FUNCTION_BLOCK COLORSENSOR_MDL (* Color sensor model *)
  (* Standard: 61499-2 *)
  (* Version 0.3, 2009-09-15, JHC, Holobloc Inc, Changed transition priorities. *)
  (* Version 0.2, 2003-12-04, JHC, Rockwell Automation, Renamed for better indexing. *)
  (* Version 0.1, 2002-11-05, JHC, Rockwell Automation, Corrected missing ST element in Algorithm REQ. *)
  (* Version 0.0, 2000-05-30, JHC, Rockwell Automation *)
  (* Compiler header: package fb.rt.dasdA1.A2; *)
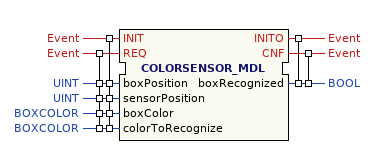
  EVENT_INPUT
    INIT WITH boxPosition, sensorPosition, boxColor, colorToRecognize; (* Initialization Request *)
    REQ WITH boxPosition, sensorPosition, colorToRecognize, boxColor; (* Normal Execution Request *)
  END_EVENT
  EVENT_OUTPUT
    INITO WITH boxRecognized; (* Initialization Confirm *)
    CNF WITH boxRecognized; (* Execution Confirmation *)
  END_EVENT
  VAR_INPUT
    boxPosition : UINT; (* Position of box in conveyor *)
    sensorPosition : UINT; (* Sensor position relative to conveyor *)
    boxColor : BOXCOLOR; (* Color of the box *)
    colorToRecognize : BOXCOLOR; (* Color which sensor will recognize *)
  END_VAR
  VAR_OUTPUT
    boxRecognized : BOOL; (* TRUE if colors and positions matches *)
  END_VAR
  VAR
    window : UINT := 10; (* Window for box position recognization *)
    windowMin : UINT;
    windowMax : UINT;
  END_VAR
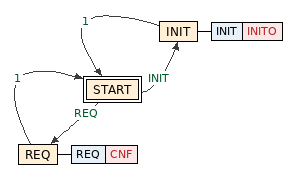
  EC_STATES
    START; (* Initial State *)
    INIT : INIT -> INITO; (* Initialization *)
    REQ : REQ -> CNF; (* Normal execution *)
  END_STATES
  EC_TRANSITIONS
    INIT TO START := 1;
    START TO REQ := REQ;
    START TO INIT := INIT;
    REQ TO START := 1;
  END_TRANSITIONS
  ALGORITHM INIT IN ST: (* Initialization algorithm *)
IF window > sensorPosition THEN
	windowMin := 0;
	windowMax := sensorPosition * 2;
ELSE
	windowMin := sensorPosition - window;
	windowMax := sensorPosition + window;
END_IF;
  END_ALGORITHM
  ALGORITHM REQ IN ST: (* Normally executed algorithm *)
IF boxPosition >= windowMin
	AND boxPosition <= windowMax
	AND boxColor = colorToRecognize
THEN
	boxRecognized := TRUE;
ELSE
	boxRecognized := FALSE;
END_IF;
  END_ALGORITHM
END_FUNCTION_BLOCK
